TYPE (* DataPanel Modules with medium IO density DI Struct + Source Address *)
  (* Version 1.0, 2026-05-28, franz *)
  PACKAGE DataPanel::io::MI::DI;
  IMPORT DataPanel::io::MI::DI::DataPanel_MI_DI::Invalid;
  IMPORT DataPanel::io::MI::const::MI::MI_00;
  DataPanel_MI_DI_S_Dual_SA : STRUCT
    u8SAMember : USINT := MI_00; (* Node SA 224..239 *)
    Up : DataPanel::io::MI::DI::DataPanel_MI_DI_S := Invalid; (* Identify the Port 1A..8B forward, up, right, clockwise *)
    Down : DataPanel::io::MI::DI::DataPanel_MI_DI_S := Invalid; (* Identify the Port 1A..8B backward, down, left, counter-clockwise *)
  END_STRUCT;
END_TYPE
